FUNCTION_BLOCK E_SEL_BOOL (* Event-driven BOOL selection *)
  (* Standard: 61499-1; Function: Math; Type: Selection; Description: BOOL selection *)
  (* Version 0.0, 2006-03-02, JHC, Holobloc Inc *)
  (* Compiler header: package fb.rt.math; *)
  (* Compiler Java Sun JDK 1.4.2 *)
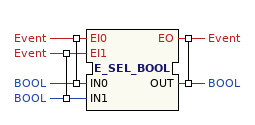
  EVENT_INPUT
    EI0 WITH IN0; (* Select INO *)
    EI1 WITH IN1; (* Select IN1 *)
  END_EVENT
  EVENT_OUTPUT
    EO WITH OUT; (* New selection event *)
  END_EVENT
  VAR_INPUT
    IN0 : BOOL; (* Selected by EI0 *)
    IN1 : BOOL; (* Selected by EI1 *)
  END_VAR
  VAR_OUTPUT
    OUT : BOOL; (* Selected value *)
  END_VAR
END_FUNCTION_BLOCK
